// TIA Portal V19 export
DATA_BLOCK "SIMATIC Ident_1"   // DB1
AUTHOR : SIMATIC
FAMILY : Ident
VERSION : 1.2
// stored: InstanceOfName TO_IDENT, OfSystemLibElement TO_IDENT, OfSystemLibVersion 1.2
TO_IDENT   // technology object, version 1.2
   // VAR
   //    HW_ID { ExternalWritable := 'False'; S7_SetPoint := 'True'} : Word;
   //    CM_CHANNEL { ExternalWritable := 'False'; S7_SetPoint := 'True'} : Int;
   //    LADDR { ExternalWritable := 'False'; S7_SetPoint := 'True'} : Word;
   //    CONFIGURATION { S7_SetPoint := 'True'} : IID_IN_PARAMETERS;
   //    DIAGNOSTIC { ExternalWritable := 'False'; S7_SetPoint := 'True'} : IID_IN_DIAGNOSTIC;
   //    STATIC { ExternalWritable := 'False'; S7_SetPoint := 'True'} : IID_IN_SYNC_TO;
   // END_VAR
BEGIN
END_DATA_BLOCK
